FUNCTION_BLOCK FB_MovingAverageFilter_3D
VAR_INPUT
    a_fNewValues : ARRAY[0..2] OF REAL; // New input values for three axes
    nNumSamples : UINT:= gvl_sensorFusion.buffersize_filter;                // Number of samples for the moving average
    bEnable : BOOL;                   // Enable flag
END_VAR

VAR_OUTPUT
    a_fAvgValues : ARRAY[0..2] OF REAL; // Output average values for three axes
    bBufferFilledX : BOOL;            // Flag indicating if the buffer for X axis is filled
    bBufferFilledY : BOOL;            // Flag indicating if the buffer for Y axis is filled
    bBufferFilledZ : BOOL;            // Flag indicating if the buffer for Z axis is filled
END_VAR

VAR_IN_OUT
    a_fSamples : ARRAY[0..2] OF ARRAY[ 0..GVL_SensorFusion.buffersize_filter-1] OF REAL; // Array of arrays to store samples for three axes
END_VAR

VAR
    fbMovingAverageX : FB_MovingAverageFilter; // Instance for X axis
    fbMovingAverageY : FB_MovingAverageFilter; // Instance for Y axis
    fbMovingAverageZ : FB_MovingAverageFilter; // Instance for Z axis
END_VAR

fbMovingAverageX(
    fInputValue := a_fNewValues[0],
    nNumSamples := nNumSamples,
    bEnable := bEnable,
    fAvgValue => a_fAvgValues[0],
    bBufferFilled => bBufferFilledX,
    a_fSamples := a_fSamples[0]
);

fbMovingAverageY(
    fInputValue := a_fNewValues[1],
    nNumSamples := nNumSamples,
    bEnable := bEnable,
    fAvgValue => a_fAvgValues[1],
    bBufferFilled => bBufferFilledY,
    a_fSamples := a_fSamples[1]
);

fbMovingAverageZ(
    fInputValue := a_fNewValues[2],
    nNumSamples := nNumSamples,
    bEnable := bEnable,
    fAvgValue => a_fAvgValues[2],
    bBufferFilled => bBufferFilledZ,
    a_fSamples := a_fSamples[2]
);

END_FUNCTION_BLOCK

(* stored: Version 1.1.0.1, ProductVersion 3.1.4024.13
   POU FB_MovingAverageFilter_3D: Id {cfc77347-1872-41de-ac52-a9ef65cd48b5}, SpecialFunc None *)
